DATA_BLOCK "Station8LoadData"
VAR
  "PLC.PartTypeID" : Int;
  "PLC.Station8RecipeNo" : Int;
  "PLC.Station8DMXCode" : String[128];
  Spare : Byte;
  "MES.ErrorCode" : Int;
  "MES.StatusBits" : DInt;
  "MES.Cycle_ID" : DInt;
  "MES.Unit_ParttypeID" : Int;
END_VAR
BEGIN
END_DATA_BLOCK
